INTERFACE ITestEventHandler EXTENDS IEventHandlerBase

METHOD OnCustomEvent
VAR_INPUT
    EventArgs : IStreamReader;
END_VAR
END_METHOD

END_INTERFACE

(* stored: Version 1.1.0.1, ProductVersion 3.1.4024.4
   Itf ITestEventHandler: Id {055a612e-0961-42c1-b0dc-25a07fda39e5}
   Method OnCustomEvent: Id {d5053930-9984-44e5-8c3a-7686797bebd5} *)
